FUNCTION_BLOCK Bunker2 (* Basic FB with empty ECC *)
  (* Standard: 61499-2 *)
  (* Version 1.0, 2021-08-03, AK121668 *)
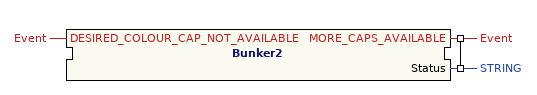
  EVENT_INPUT
    DESIRED_COLOUR_CAP_NOT_AVAILABLE; (* start feeding bunker *)
  END_EVENT
  EVENT_OUTPUT
    MORE_CAPS_AVAILABLE WITH Status; (* feeding is DONE *)
  END_EVENT
  VAR_OUTPUT
    Status : STRING; (* Current Status of Bunker *)
  END_VAR
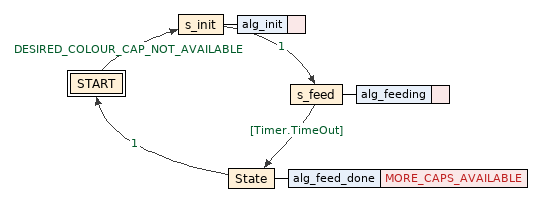
  EC_STATES
    START; (* Initial State *)
    s_feed : alg_feeding;
    State : alg_feed_done -> MORE_CAPS_AVAILABLE;
    s_init : alg_init;
  END_STATES
  EC_TRANSITIONS
    s_feed TO State := [Timer.TimeOut];
    State TO START := 1;
    START TO s_init := DESIRED_COLOUR_CAP_NOT_AVAILABLE;
    s_init TO s_feed := 1;
  END_TRANSITIONS
  ALGORITHM alg_init IN ST: (* // *)
//
Timer.DT := T#10s;
Status :='init mode';
  END_ALGORITHM
  ALGORITHM alg_feeding IN ST: (* // *)
//
Status :='feeding now';
  END_ALGORITHM
  ALGORITHM alg_feed_done IN ST: (* // *)
//
Status :='feeding Done';
  END_ALGORITHM
END_FUNCTION_BLOCK
